// TwinCAT 3 PLC project PlcMatt
// ProgramVersion: 3.1.4026.23
// libraries:
//   Tc2_Standard, * (Beckhoff Automation GmbH)
//   Tc2_System, * (Beckhoff Automation GmbH)
// project tree:
//   DUTs/CMMT_AS/ E_CMMT_BrakeStatus.TcDUT, ST_CMMT_DriveToPlc.TcDUT, ST_CMMT_PlcToDrive.TcDUT
//   DUTs/ E_MotorStatus.TcDUT, ST_WarningBits.TcDUT, U_ARRAY_64.TcDUT, U_UNIONN.TcDUT
//   DUTs/MX2/ MX2_Inputs.TcDUT, MX2_Outputs.TcDUT, ST_MX2_CommandBits.TcDUT, ST_MX2_Outputs.TcDUT, U_MX2_CommandWord.TcDUT
//   GVLs/ GVL.TcGVL
//   / PlcTask.TcTTO
//   POUs/FBs/ FB_CMMT_BrakeControl.TcPOU, FB_Motor.TcPOU, FB_TestPopup.TcPOU
//   POUs/ MAIN.TcPOU, PRG_CMMT_AS.TcPOU, PRG_MX2_Testing.TcPOU
// real-time tasks:
//   TASK PlcTask: cycle T#100000us, priority 20, ADS port 350
// I/O:
//   DEVICE LAN ECT (EtherCAT) (disabled), AmsNetId 10.10.20.20.2.1
//     Box 1 (3G3AX-MX2-ECT) [3G3AX-MX2-ECT EtherCAT Communication Unit for 3G3MX2]
//     Drive 2 (CMMT-AS) [CMMT-AS]
// variable links:
//   PlcMatt/PlcMatt Instance <-> LAN ECT (EtherCAT)/Box 1 (3G3AX-MX2-ECT)
//     PlcTask Inputs/GVL.MX2_UDTs_Check._3G3AX_MX2_ECT_Input/InfoData_AdsAddr <-> InfoData/AdsAddr
//     PlcTask Inputs/GVL.MX2_UDTs_Check._3G3AX_MX2_ECT_Input/InfoData_State <-> InfoData/State
//     PlcTask Inputs/GVL.MX2_UDTs_Check._3G3AX_MX2_ECT_Input/WcState_InputToggle <-> WcState/InputToggle
//     PlcTask Inputs/GVL.MX2_UDTs_Check._3G3AX_MX2_ECT_Input/WcState_WcState <-> WcState/WcState

CONFIGURATION PlcMatt
    RESOURCE PLC ON TwinCAT3
        TASK PlcTask(INTERVAL := T#100000us, PRIORITY := 20);
        PROGRAM MAIN WITH PlcTask : MAIN;
    END_RESOURCE
END_CONFIGURATION

// ---- DUTs/CMMT_AS/E_CMMT_BrakeStatus.TcDUT
{attribute 'qualified_only'}
{attribute 'strict'}
{attribute 'to_string'}
TYPE E_CMMT_BrakeStatus :
(
    Closed  := 0,    // Brake is reported closed/applied
    Open    := 1,    // Brake is reported open/released
    Opening := 2,    // Brake is currently opening
    Closing := 3,    // Brake is currently closing

    Invalid := 4     // Value received from drive is not recognised
);
END_TYPE

// ---- DUTs/CMMT_AS/ST_CMMT_DriveToPlc.TcDUT
{attribute 'pack_mode' := '1'}
TYPE ST_CMMT_DriveToPlc :
STRUCT
    wStatusword               : UINT;     // 6041:00
    nModesOfOperationDisplay  : SINT;     // 6061:00
    diPositionActual          : DINT;     // 6064:00
    diVelocityActual          : DINT;     // 606C:00
    iTorqueActual             : INT;      // 6077:00
    byPadding                 : BYTE;

    udiBrake1Status           : UDINT;    // 2150:05
END_STRUCT
END_TYPE

// ---- DUTs/CMMT_AS/ST_CMMT_PlcToDrive.TcDUT
{attribute 'pack_mode' := '1'}
TYPE ST_CMMT_PlcToDrive :
STRUCT
    wControlword              : UINT;     // 6040:00
    nModesOfOperation         : SINT;     // 6060:00
    diTargetPosition          : DINT;     // 607A:00
    udiProfileVelocity        : UDINT;    // 6081:00
    diTargetVelocity          : DINT;     // 60FF:00
    iTargetTorque             : INT;      // 6071:00
    diVelocityOffset          : DINT;     // 60B1:00
    iTorqueOffset             : INT;      // 60B2:00
    byPadding                 : BYTE;

    udiProfileAcceleration    : UDINT;    // 6083:00
    udiProfileDeceleration    : UDINT;    // 6084:00
    udiDigitalOutputs         : UDINT;    // 60FE:01
    udiDigitalOutputsMask     : UDINT;    // 60FE:02
END_STRUCT
END_TYPE

// ---- DUTs/E_MotorStatus.TcDUT
{attribute 'qualified_only'}
{attribute 'strict'}
{attribute 'to_string'}

TYPE E_MotorStatus :
(
    eMotorStatus_NotReady := 0,
    eMotorStatus_Ready := 1,
    eMotorStatus_Stopped := 2,
    eMotorStatus_Starting := 3,
    eMotorStatus_Running := 4,
    eMotorStatus_Stopping := 5,
    eMotorStatus_Fault := 6,
    eMotorStatus_StartTimeout := 7,
    eMotorStatus_StopTimeout := 8,
    eMotorStatus_ExternalFault := 9,
    eMotorStatus_InterlockFault := 10
);
END_TYPE

// ---- DUTs/MX2/MX2_Inputs.TcDUT
{attribute 'TcTypeSystem'}
{attribute 'GUID' := '33A1B596-0D78-759C-A1DE-33D224F34F3C'}
TYPE MX2_Inputs :
	STRUCT
		{attribute 'GUID' := '33A1B597-0D78-759C-A1DE-33D224F34F3C'}
		_3G3AX_MX2_ECT_Input AT %I* : _3G3AX_MX2_ECT_I_A841956B;
	END_STRUCT
END_TYPE

// ---- DUTs/MX2/MX2_Outputs.TcDUT
{attribute 'TcTypeSystem'}
TYPE MX2_Outputs :
	STRUCT
		_3G3AX_MX2_ECT_Output AT %Q* : ST_MX2_Outputs;
	END_STRUCT
END_TYPE

// ---- DUTs/MX2/ST_MX2_CommandBits.TcDUT
TYPE ST_MX2_CommandBits :
STRUCT
    bForwardRun     : BIT;  // Bit 0: forward / position start
    bReverseRun     : BIT;  // Bit 1: reverse / position start

    bReserved02     : BIT;  // Bit 2
    bReserved03     : BIT;  // Bit 3
    bReserved04     : BIT;  // Bit 4
    bReserved05     : BIT;  // Bit 5
    bReserved06     : BIT;  // Bit 6

    bFaultReset     : BIT;  // Bit 7

    bReserved08     : BIT;  // Bit 8
    bReserved09     : BIT;  // Bit 9
    bReserved10     : BIT;  // Bit 10
    bReserved11     : BIT;  // Bit 11
    bReserved12     : BIT;  // Bit 12
    bReserved13     : BIT;  // Bit 13
    bReserved14     : BIT;  // Bit 14
    bReserved15     : BIT;  // Bit 15
END_STRUCT
END_TYPE

// ---- DUTs/MX2/ST_MX2_Outputs.TcDUT
{attribute 'pack_mode' := '1'}
TYPE ST_MX2_Outputs :
STRUCT
    uiCommand               : UINT;   // Offset 0,  2 bytes
    uiFrequencyReference    : UINT;   // Offset 2,  2 bytes
    diTargetPosition        : DINT;   // Offset 4,  4 bytes, P060
    udiAccelerationTime     : UDINT;  // Offset 8,  4 bytes, F002
    udiDecelerationTime     : UDINT;  // Offset 12, 4 bytes, F003
    uiCoilData0             : UINT;   // Offset 16, 2 bytes
    uiOutputTerminalSetting : UINT;   // Offset 18, 2 bytes
END_STRUCT
END_TYPE

// ---- DUTs/MX2/U_MX2_CommandWord.TcDUT
TYPE U_MX2_CommandWord :
UNION
    wValue : WORD;
    stBits : ST_MX2_CommandBits;
END_UNION
END_TYPE

// ---- DUTs/ST_WarningBits.TcDUT
TYPE ST_WarningBits :
STRUCT
    bEmergencyStop        : BIT; // Bit 0  - Emergency stop active
    bSafetyGateOpen       : BIT; // Bit 1  - Safety gate is open
    bAirPressureLow       : BIT; // Bit 2  - Pneumatic pressure too low
    bDriveFault           : BIT; // Bit 3  - Servo drive reports a fault
    bMotorOverload        : BIT; // Bit 4  - Motor overload detected
    bAxisNotHomed         : BIT; // Bit 5  - Axis requires homing
    bPositionTimeout      : BIT; // Bit 6  - Positioning timeout
    bCommunicationFault   : BIT; // Bit 7  - Fieldbus communication fault

    bSensor01Fault        : BIT; // Bit 8  - Sensor 01 not detected
    bSensor02Fault        : BIT; // Bit 9  - Sensor 02 not detected
    bReserved10           : BIT; // Bit 10 - Reserved
    bReserved11           : BIT; // Bit 11 - Reserved
    bReserved12           : BIT; // Bit 12 - Reserved
    bReserved13           : BIT; // Bit 13 - Reserved
    bReserved14           : BIT; // Bit 14 - Reserved
    bReserved15           : BIT; // Bit 15 - Reserved
	
	test : word;

    Sensor01Fault        : BIT; // Bit 8  - Sensor 01 not detected
    Sensor02Fault        : BIT; // Bit 9  - Sensor 02 not detected
    Reserved10           : BIT; // Bit 10 - Reserved
    Reserved11           : BIT; // Bit 11 - Reserved
    Reserved12           : BIT; // Bit 12 - Reserved
    Reserved13           : BIT; // Bit 13 - Reserved
    Reserved14           : BIT; // Bit 14 - Reserved
    Reserved15           : BIT; // Bit 15 - Reserved
    // Continue through bit 63...
END_STRUCT
END_TYPE

// ---- DUTs/U_ARRAY_64.TcDUT
TYPE U_ARRAY_64 :
UNION
	
	WrnAryWord : ARRAY[0..3] OF WORD;
	WrnAryDWord : ARRAY[0..1] OF DWORD;
	WrnAryBit : ARRAY[0..63] OF BOOL;
	stTest: ST_WarningBits;
END_UNION
END_TYPE

// ---- DUTs/U_UNIONN.TcDUT
TYPE U_UNIONN :
UNION
	
	WrnAryByte : ARRAY[0..7] OF BYTE;
	WrnAryWord : ARRAY[0..3] OF WORD;
	WrnAryDWord : ARRAY[0..1] OF DWORD;
	stTest: ST_WarningBits;
END_UNION
END_TYPE

// ---- GVLs/GVL.TcGVL
{attribute 'qualified_only'}
VAR_GLOBAL
	
Motor1 : FB_Motor;
Motor2 : FB_Motor;

PopupTest1 : FB_TestPopup;
PopupTest2 : FB_TestPopup;


MX2_UDTs_Check : _3G3AX_MX2_ECT_A841956B;
MX2_Outputs : MX2_Outputs;


END_VAR

VAR_GLOBAL PERSISTENT
    nCycleCount : DINT := 0; 
    fTargetTemperature : REAL := 25.5;
    bMachineFault : BOOL := FALSE;
END_VAR

// ---- POUs/MAIN.TcPOU
PROGRAM MAIN
VAR
	bTest : BOOL;
	i : LINT;
	iTest : LINT :=5;
		
	Motor1 : REFERENCE TO FB_Motor;
	Motor2 : REFERENCE TO FB_Motor;	
	
	PopupTest1 : REFERENCE TO FB_TestPopup;
	PopupTest2 : REFERENCE TO FB_TestPopup;
	
	WrnAry : ARRAY[0..63] OF BOOL;
	Alr1Ary : ARRAY[0..63] OF BOOL;
	Alr2Ary : ARRAY[0..63] OF BOOL;
	Alr3Ary : ARRAY[0..63] OF BOOL;
	
	uAlarms : U_ARRAY_64;
	uUnionTest : U_UNIONN;
	
	bTest_MX2 : BOOL;
	
END_VAR


Motor1 REF= GVL.Motor1;
Motor2 REF= GVL.Motor2;


PopupTest1 REF= GVL.PopupTest1;
PopupTest2 REF= GVL.PopupTest2;


iTest := iTest + 1;

FOR i := 0 TO  iTest DO
	
	;
	//iTest := iTest + 1;
END_FOR;


Motor1();
Motor2();

PopupTest1();
PopupTest2();


bTest_MX2 := GVL.MX2_UDTs_Check._3G3AX_MX2_ECT_Input.WcState_WcState;

//uAlarms.WrnAryBit := WrnAry;

END_PROGRAM

// ---- POUs/FBs/FB_Motor.TcPOU
FUNCTION_BLOCK FB_Motor
VAR_INPUT
    i_bEnable           : BOOL;
    i_bAutoMode         : BOOL;
    i_bManMode          : BOOL;

    i_bAutoStart        : BOOL;
    i_bManStart         : BOOL;
    i_bStop             : BOOL;
    i_bReset            : BOOL;

    i_bPermissive       : BOOL := TRUE;
    i_bInterlockOk      : BOOL := TRUE;
    i_bEmergencyOk      : BOOL := TRUE;

    i_bRunFeedback      : BOOL;
    i_bExternalFault    : BOOL;

    i_tStartTimeout     : TIME := T#5S;
    i_tStopTimeout      : TIME := T#5S;
END_VAR

VAR_OUTPUT
    o_bRunCmd           : BOOL;

    o_bReady            : BOOL;
    o_bRunning          : BOOL;
    o_bStopped          : BOOL;
    o_bStarting         : BOOL;
    o_bStopping         : BOOL;
    o_bFault            : BOOL;

    o_bStartTimeout     : BOOL;
    o_bStopTimeout      : BOOL;
    o_bInterlockFault   : BOOL;
    o_bExternalFault    : BOOL;

    o_eStatus           : E_MotorStatus;
END_VAR

VAR
    bStartRequest       : BOOL;
    bCanRun             : BOOL;
    bFaultLatched       : BOOL;

    tonStartTimeout     : TON;
    tonStopTimeout      : TON;

    rtrigReset          : R_TRIG;
END_VAR



// ======================================================
// Reset edge
// ======================================================
rtrigReset(CLK := i_bReset);


// ======================================================
// Conditions
// ======================================================
bCanRun :=
    i_bEnable AND
    i_bPermissive AND
    i_bInterlockOk AND
    i_bEmergencyOk AND
    NOT bFaultLatched;


// ======================================================
// Start request
// ======================================================
bStartRequest :=
    (i_bAutoMode AND i_bAutoStart) OR
    (i_bManMode AND i_bManStart);


// ======================================================
// Fault handling
// ======================================================
o_bExternalFault := i_bExternalFault;

IF i_bExternalFault THEN
    bFaultLatched := TRUE;
END_IF

IF NOT i_bInterlockOk THEN
    o_bInterlockFault := TRUE;
    bFaultLatched := TRUE;
END_IF

IF o_bStartTimeout THEN
    bFaultLatched := TRUE;
END_IF

IF o_bStopTimeout THEN
    bFaultLatched := TRUE;
END_IF

IF rtrigReset.Q THEN
    IF NOT i_bExternalFault
    AND i_bInterlockOk
    AND i_bEmergencyOk THEN
        bFaultLatched := FALSE;
        o_bStartTimeout := FALSE;
        o_bStopTimeout := FALSE;
        o_bInterlockFault := FALSE;
    END_IF
END_IF


// ======================================================
// Run command
// ======================================================
IF i_bStop OR NOT i_bEnable OR bFaultLatched THEN
    o_bRunCmd := FALSE;
ELSIF bCanRun AND bStartRequest THEN
    o_bRunCmd := TRUE;
END_IF


// ======================================================
// Timers
// ======================================================
tonStartTimeout(
    IN := o_bRunCmd AND NOT i_bRunFeedback,
    PT := i_tStartTimeout
);

tonStopTimeout(
    IN := NOT o_bRunCmd AND i_bRunFeedback,
    PT := i_tStopTimeout
);

IF tonStartTimeout.Q THEN
    o_bStartTimeout := TRUE;
END_IF

IF tonStopTimeout.Q THEN
    o_bStopTimeout := TRUE;
END_IF


// ======================================================
// Status bits
// ======================================================
o_bFault    := bFaultLatched;
o_bRunning  := i_bRunFeedback AND NOT o_bFault;
o_bStopped  := NOT i_bRunFeedback AND NOT o_bRunCmd AND NOT o_bFault;
o_bStarting := o_bRunCmd AND NOT i_bRunFeedback AND NOT o_bFault;
o_bStopping := NOT o_bRunCmd AND i_bRunFeedback AND NOT o_bFault;
o_bReady    := bCanRun AND NOT o_bRunCmd AND NOT i_bRunFeedback;


// ======================================================
// ENUM status
// ======================================================
IF o_bExternalFault THEN
    o_eStatus := E_MotorStatus.eMotorStatus_ExternalFault;

ELSIF o_bInterlockFault THEN
    o_eStatus := E_MotorStatus.eMotorStatus_InterlockFault;

ELSIF o_bStartTimeout THEN
    o_eStatus := E_MotorStatus.eMotorStatus_StartTimeout;

ELSIF o_bStopTimeout THEN
    o_eStatus := E_MotorStatus.eMotorStatus_StopTimeout;

ELSIF o_bFault THEN
    o_eStatus := E_MotorStatus.eMotorStatus_Fault;

ELSIF o_bRunning THEN
    o_eStatus := E_MotorStatus.eMotorStatus_Running;

ELSIF o_bStarting THEN
    o_eStatus := E_MotorStatus.eMotorStatus_Starting;

ELSIF o_bStopping THEN
    o_eStatus := E_MotorStatus.eMotorStatus_Stopping;

ELSIF o_bReady THEN
    o_eStatus := E_MotorStatus.eMotorStatus_Ready;

ELSIF o_bStopped THEN
    o_eStatus := E_MotorStatus.eMotorStatus_Stopped;

ELSE
    o_eStatus := E_MotorStatus.eMotorStatus_NotReady;
END_IF

END_FUNCTION_BLOCK

// ---- POUs/FBs/FB_TestPopup.TcPOU
FUNCTION_BLOCK FB_TestPopup
VAR_INPUT
	i_PopupReq : BOOL;// 1=Popup, 0=No popup
END_VAR
VAR_OUTPUT
	o_PopupResult : BOOL;
END_VAR
VAR
	bPopupResult : BOOL;
	iPopupN : INT;
	bButtonPressed : BOOL;
	bPopupOK : BOOL;
	
END_VAR

o_PopupResult := bPopupResult;

END_FUNCTION_BLOCK

// ---- POUs/FBs/FB_CMMT_BrakeControl.TcPOU
FUNCTION_BLOCK FB_CMMT_BrakeControl
VAR_INPUT
    (*
        Enables control of the brake-release-request PDO bit.

        FALSE:
            The FB clears bit 0 of the output mask.
            The PLC does not request control of the brake-release bit.

        TRUE:
            The FB sets bit 0 of 60FE:02.
            The PLC controls bit 0 of 60FE:01.

        For a manual/service brake-release function, this input would
        normally be enabled only while the machine is in an authorised
        service or commissioning mode.
    *)
    i_bEnableManualBrakeControl : BOOL;


    (*
        Operator or application request to release the holding brake.

        FALSE:
            No manual release request.

        TRUE:
            Request the CMMT to release/open the holding brake.

        This input does not bypass i_bReleasePermitted.
    *)
    i_bManualBrakeRelease : BOOL;


    (*
        Application interlock permitting brake release.

        Suggested conditions for a vertical axis include:

            - Safety system permits movement
            - Axis is mechanically supported, or motor torque is established
            - Machine is in an authorised operating mode
            - No active brake-related fault
            - No conflicting stop or emergency command

        The FB only issues the release request when this input is TRUE.
    *)
    i_bReleasePermitted : BOOL;


    (*
        Raw brake status received from object 2150:05.

        Expected values:

            0 = Brake closed
            1 = Brake open
            2 = Brake opening
            3 = Brake closing
    *)
    i_udiBrakeStatusRaw : UDINT;
END_VAR


VAR_IN_OUT
    (*
        Object 60FE:01 — Digital outputs.

        Only bit 0 is modified by this FB.
        All other bits are preserved.
    *)
    io_udiDigitalOutputs : UDINT;


    (*
        Object 60FE:02 — Digital output mask.

        Only bit 0 is modified by this FB.
        All other mask bits are preserved.
    *)
    io_udiDigitalOutputsMask : UDINT;
END_VAR


VAR_OUTPUT
    (*
        TRUE when the PLC currently owns the brake-release bit and is
        actively sending a release request.
    *)
    o_bReleaseRequestActive : BOOL;


    (*
        Decoded brake status.
    *)
    o_eBrakeStatus : E_CMMT_BrakeStatus;


    (*
        Individual status outputs for simple use in application logic
        and HMI displays.
    *)
    o_bBrakeClosed  : BOOL;
    o_bBrakeOpen    : BOOL;
    o_bBrakeOpening : BOOL;
    o_bBrakeClosing : BOOL;


    (*
        TRUE while the brake is either opening or closing.
    *)
    o_bBrakeTransitioning : BOOL;


    (*
        TRUE when 2150:05 contains one of the documented values 0...3.

        FALSE means that an unexpected value was received.
    *)
    o_bBrakeStatusValid : BOOL;


    (*
        TRUE when the operator requested brake release, but an application
        interlock prevented the request from being sent.
    *)
    o_bReleaseRequestBlocked : BOOL;
END_VAR


VAR
    (*
        Final internally calculated release request.

        The EtherCAT command is only issued when all three conditions
        are TRUE.
    *)
    bReleaseRequest : BOOL;
END_VAR


VAR CONSTANT
    (*
        Bit mask for bit 0.

        This bit is used in both:

            60FE:01 Digital outputs
            60FE:02 Digital output mask
    *)
    C_UDI_BRAKE_RELEASE : UDINT := 16#00000001;
END_VAR


(*
    =====================================================================
    CALCULATE THE FINAL BRAKE-RELEASE REQUEST
    =====================================================================

    The request is accepted only when:

        1. Manual brake control is enabled.
        2. A brake-release request is present.
        3. The application permits brake release.
*)
bReleaseRequest :=
    i_bEnableManualBrakeControl
    AND i_bManualBrakeRelease
    AND i_bReleasePermitted;


(*
    Indicate when the requested operation has been blocked by an
    application interlock.

    This can be displayed on the HMI to explain why pressing the
    brake-release button did not release the brake.
*)
o_bReleaseRequestBlocked :=
    i_bEnableManualBrakeControl
    AND i_bManualBrakeRelease
    AND NOT i_bReleasePermitted;


(*
    =====================================================================
    CONTROL 60FE:02 — DIGITAL OUTPUT MASK
    =====================================================================

    Setting bit 0 in the mask gives the fieldbus/PLC control over
    bit 0 of 60FE:01.

    OR is used instead of direct assignment so that any other output-mask
    bits used elsewhere in the application are not overwritten.
*)
IF i_bEnableManualBrakeControl THEN

    io_udiDigitalOutputsMask :=
        io_udiDigitalOutputsMask OR C_UDI_BRAKE_RELEASE;

ELSE

    (*
        Remove PLC control of the brake-release-request bit.

        AND NOT clears only bit 0 and preserves all other mask bits.
    *)
    io_udiDigitalOutputsMask :=
        io_udiDigitalOutputsMask AND (NOT C_UDI_BRAKE_RELEASE);

END_IF


(*
    =====================================================================
    CONTROL 60FE:01 — BRAKE RELEASE REQUEST
    =====================================================================

    Bit 0 = 1:
        Request the holding brake to open/release.

    Bit 0 = 0:
        Remove the manual release request.

    OR and AND NOT are used so that all other digital-output bits remain
    unchanged.
*)
IF bReleaseRequest THEN

    io_udiDigitalOutputs :=
        io_udiDigitalOutputs OR C_UDI_BRAKE_RELEASE;

ELSE

    io_udiDigitalOutputs :=
        io_udiDigitalOutputs AND (NOT C_UDI_BRAKE_RELEASE);

END_IF


(*
    Confirm the command that is actually present in the PDO data.

    Both conditions must be true:

        - Output mask bit 0 is enabled.
        - Digital output bit 0 is set.
*)
o_bReleaseRequestActive :=
    ((io_udiDigitalOutputsMask AND C_UDI_BRAKE_RELEASE) <> 0)
    AND
    ((io_udiDigitalOutputs AND C_UDI_BRAKE_RELEASE) <> 0);


(*
    =====================================================================
    INITIALISE BRAKE STATUS OUTPUTS
    =====================================================================

    Outputs are reset every PLC cycle before decoding the status.

    This prevents an old TRUE state from remaining latched when the
    drive changes to another brake state.
*)
o_eBrakeStatus          := E_CMMT_BrakeStatus.Invalid;

o_bBrakeClosed          := FALSE;
o_bBrakeOpen            := FALSE;
o_bBrakeOpening         := FALSE;
o_bBrakeClosing         := FALSE;
o_bBrakeTransitioning   := FALSE;
o_bBrakeStatusValid     := FALSE;


(*
    =====================================================================
    DECODE 2150:05 — HOLDING BRAKE 1 STATUS
    =====================================================================

        Value 0:
            Brake closed/applied.

        Value 1:
            Brake open/released.

        Value 2:
            Brake opening.

        Value 3:
            Brake closing.

    The opening and closing states are transitional states.
*)
CASE i_udiBrakeStatusRaw OF

    0:
        (*
            Brake closed/applied.

            The drive reports that the brake-control sequence has reached
            the closed state.
        *)
        o_eBrakeStatus      := E_CMMT_BrakeStatus.Closed;
        o_bBrakeClosed      := TRUE;
        o_bBrakeStatusValid := TRUE;


    1:
        (*
            Brake open/released.

            The drive reports that the brake-control sequence has reached
            the open state.
        *)
        o_eBrakeStatus      := E_CMMT_BrakeStatus.Open;
        o_bBrakeOpen        := TRUE;
        o_bBrakeStatusValid := TRUE;


    2:
        (*
            Brake opening.

            The CMMT is currently executing the configured brake-opening
            sequence or brake-release delay.
        *)
        o_eBrakeStatus          := E_CMMT_BrakeStatus.Opening;
        o_bBrakeOpening         := TRUE;
        o_bBrakeTransitioning   := TRUE;
        o_bBrakeStatusValid     := TRUE;


    3:
        (*
            Brake closing.

            The CMMT is currently executing the configured brake-closing
            sequence or brake-application delay.
        *)
        o_eBrakeStatus          := E_CMMT_BrakeStatus.Closing;
        o_bBrakeClosing         := TRUE;
        o_bBrakeTransitioning   := TRUE;
        o_bBrakeStatusValid     := TRUE;


ELSE
    (*
        Unexpected or unsupported value.

        This can indicate:

            - Incorrect PDO mapping
            - Incorrect data type
            - Incorrect byte alignment
            - Firmware/object-version mismatch
            - Invalid data while EtherCAT is not operational
    *)
    o_eBrakeStatus      := E_CMMT_BrakeStatus.Invalid;
    o_bBrakeStatusValid := FALSE;

END_CASE

END_FUNCTION_BLOCK

// ---- POUs/PRG_CMMT_AS.TcPOU
PROGRAM PRG_CMMT_AS
VAR
	
	stCMMT_In : ST_CMMT_DriveToPlc;
	stCMMT_Out : ST_CMMT_PlcToDrive;


    fbCMMTBrake : FB_CMMT_BrakeControl;

    // Command from HMI or service controls.
    bManualBrakeRelease : BOOL;

    // Recommended release interlocks.
    bServiceMode               : BOOL;
    bSafetyPermitsRelease      : BOOL;
    bAxisMechanicallySupported : BOOL;



END_VAR

(*


// EtherCAT DIP Switch Configuration
SW1    SW2    SW3
 0      1      0
OFF     ON    OFF



Beckhoff EtherCAT master
          │
          ▼
CMMT-AS [XF1 IN]
CMMT-AS [XF2 OUT]
          │
          ▼
Next EtherCAT slave

*)

(*
CMMT-AS — CiA 402 motion start behaviour

```
There is no separate universal "Start" PDO.

The function of Controlword bits 4...6 depends on the operating
mode selected with object 6060h "Modes of operation".

Always wait until object 6061h "Modes of operation display"
confirms the requested mode before issuing a motion command.

---------------------------------------------------------------
MODE 1 — PROFILE POSITION
---------------------------------------------------------------

6060h := 1

The CMMT generates the position trajectory internally.

Before starting:
  1. Write Target position 607Ah.
  2. Write Profile velocity 6081h.
  3. Write acceleration/deceleration, when required.
  4. Make sure Controlword bit 4 is FALSE.

Start positioning with a rising edge of Controlword bit 4:

    Bit 4: FALSE -> TRUE

Relevant Controlword bits:
  Bit 4 = New set-point / start positioning
  Bit 5 = Change set-point immediately
  Bit 6 = 0: absolute position
          1: relative position
  Bit 8 = Halt

Position-command handshake:
  1. Set bit 4.
  2. Wait for Statusword bit 12 = TRUE
     (set-point acknowledged).
  3. Clear Controlword bit 4.
  4. Wait for Statusword bit 12 = FALSE.
  5. Wait for Statusword bit 10 = TRUE
     (target reached).

Merely changing Target position 607Ah does not start a movement.
A new FALSE-to-TRUE transition of Controlword bit 4 is required
for every new positioning command.

---------------------------------------------------------------
MODE 3 — PROFILE VELOCITY / JOG
---------------------------------------------------------------

6060h := 3

There is no separate Start bit in Profile Velocity mode.

Movement is controlled directly by Target velocity 60FFh:

    Target velocity > 0  : move in positive direction
    Target velocity < 0  : move in negative direction
    Target velocity = 0  : decelerate to standstill

Therefore, jogging is active while a non-zero signed target
velocity is being commanded.

Controlword bit 8 may be used to request Halt.

Before changing from Profile Velocity to another mode:
  1. Command Target velocity := 0.
  2. Wait until actual velocity is approximately zero.
  3. Select the new mode in 6060h.
  4. Wait until 6061h confirms the new mode.

---------------------------------------------------------------
MODE 6 — HOMING
---------------------------------------------------------------

6060h := 6

The homing method, direction, speeds and acceleration are
configured in Festo Automation Suite or through parameters.

Start homing with a rising edge of Controlword bit 4:

    Bit 4: FALSE -> TRUE

Relevant Statusword bits:
  Bit 12 = Homing attained
  Bit 13 = Homing error

Keep the homing-start command active while homing is running,
then clear Controlword bit 4 after homing has completed or failed.

---------------------------------------------------------------
IMPORTANT
---------------------------------------------------------------

Controlword bits 4...6 must never be interpreted without first
considering the active operating mode.

The same physical bit can have a different function in:
  Mode 1: Profile Position
  Mode 3: Profile Velocity
  Mode 6: Homing
  Mode 8: Cyclic Synchronous Position

Mode 8 must not be used for simple direct PLC positioning unless
the PLC continuously generates cyclic trajectory set-points.
```

*)







(*

Reading brake status The values of 2150:05 are: Value Meaning 0 Brake closed 1 Brake open 2 Brake opening 3 Brake closing

*)



(*
    =====================================================================
    CMMT-AS HOLDING BRAKE CONTROL
    =====================================================================

    EtherCAT / CoE objects used:

        60FE:01    Digital outputs
        60FE:02    Digital output mask
        2150:05    Holding brake 1 status

    Brake release command:

        60FE:01 bit 0 = 1
            Request the holding brake to release/open.

        60FE:01 bit 0 = 0
            Remove the holding-brake release request.

    Output control mask:

        60FE:02 bit 0 = 1
            The fieldbus/PLC controls bit 0 of 60FE:01.

        60FE:02 bit 0 = 0
            The fieldbus/PLC does not control this output bit.

    IMPORTANT:

    The command is called "Brake Release Request" because the PLC is
    requesting that the CMMT releases the brake. It is not direct proof
    that the mechanical brake is physically open.

    For a vertical axis, releasing the brake without motor torque or
    mechanical support can allow the load to fall.

    The manual brake-release command should normally be restricted to
    commissioning, maintenance or service operation.

    During normal automatic motion, the CMMT should normally coordinate:

        Motor torque enabled
        -> brake released
        -> movement allowed

    and:

        Movement stopped
        -> brake applied
        -> motor torque disabled
    =====================================================================
*)





(*
    Example for a vertical axis.

    The brake release is permitted only when:

        - The machine is in service mode.
        - The safety system permits the operation.
        - The vertical load is mechanically supported.

    Replace these conditions with the interlocks appropriate for your
    machine risk assessment.
*)
fbCMMTBrake(
    i_bEnableManualBrakeControl := bServiceMode,

    i_bManualBrakeRelease       := bManualBrakeRelease,

    i_bReleasePermitted         :=
        bSafetyPermitsRelease
        AND bAxisMechanicallySupported,

    // Object 2150:05 from the CMMT input PDO.
    i_udiBrakeStatusRaw         := stCMMT_In.udiBrake1Status,

    // Objects 60FE:01 and 60FE:02 in the CMMT output PDO.
    io_udiDigitalOutputs        := stCMMT_Out.udiDigitalOutputs,
    io_udiDigitalOutputsMask    := stCMMT_Out.udiDigitalOutputsMask
);

END_PROGRAM

// ---- POUs/PRG_MX2_Testing.TcPOU
PROGRAM PRG_MX2_Testing
VAR
END_VAR



(*



Notes for positioning


A001 = 04
A002 = 04
C102 = 03
P012 = 02

A003 = motor base frequency
A004 = maximum allowed frequency
A082 = motor rated voltage
H003 = motor capacity
H004 = motor pole number
H007 = motor rated current
A044 = 03

P003 = 01
P004 = 01
P011 = encoder PPR
C007 = 85

A051 = 00
P014 = tune
P015 = tune
P017 = tune
P060 = target position, or written by PDO
P072 = forward software limit
P073 = reverse software limit
P075 = 00

C021 = 23


// How to switch to jogging (speed mode) during Simple position Control

P012 = 02    Simple position control enabled
P075 = 00    Limit mode; SPD does not work with P075 = 01
A001 = 04    Frequency reference from EtherCAT option
A002 = 04    RUN command from EtherCAT option

C001…C007 = 73    SPD: Speed/Position switching (then write this to multi function inputs)

SPD = manual speed/jog mode
SPD OFF = simple position mode


*)

END_PROGRAM
